// Mitsubishi GX Works2 project: project_cclinkmodules   PLC: Q04UDEH

TYPE D_QJ61BT11N_IN : STRUCT
  x0ModuleError : BOOL;  (* This signal indicates whether the module is normal or faulty,True=Error *)
  x1HostDataOK : BOOL;  (* This signal indicates the data link status of the host station,True=Data Link in Process *)
  x2NotUsed : BOOL;
  x3OtherStLink : BOOL;  (* This signal indicates the data link status of other stations,True= Have Fautly Station *)
  x4NotUsed : BOOL;
  x5NotUsed : BOOL;
  x6NotUsed : BOOL;
  x7NotUsed : BOOL;
  x8NotUsed : BOOL;
  x9NotUsed : BOOL;
  xANotUsed : BOOL;
  xBNotUsed : BOOL;
  xCNotUsed : BOOL;
  xDNotUsed : BOOL;
  xENotUsed : BOOL;
  xFReady : BOOL;  (* This signal indicates whether the module is ready to operate,True=Ready *)
  x10NotUsed : BOOL;
  x11NotUsed : BOOL;
  x12NotUsed : BOOL;
  x13NotUsed : BOOL;
  x14NotUsed : BOOL;
  x15NotUsed : BOOL;
  x16NotUsed : BOOL;
  x17NotUsed : BOOL;
  x18NotUsed : BOOL;
  x19NotUsed : BOOL;
  x1ANotUsed : BOOL;
  x1BNotUsed : BOOL;
  x1CNotUsed : BOOL;
  x1DNotUsed : BOOL;
  x1ENotUsed : BOOL;
  x1FNotUsed : BOOL;
END_STRUCT END_TYPE

TYPE D_Wago_750_325_SystemArea_X : STRUCT
  x0Reserved : BOOL;
  x1Reserved : BOOL;
  x2Reserved : BOOL;
  x3Reserved : BOOL;
  x4Reserved : BOOL;
  x5Reserved : BOOL;
  x6Reserved : BOOL;
  x7Reserved : BOOL;
  x8InitDataReq : BOOL;
  x9InitDataOK : BOOL;
  xAErrorStatus : BOOL;
  xBStationRdy : BOOL;
  xCReserved : BOOL;
  xDReserved : BOOL;
  xEReserved : BOOL;
  xFReserved : BOOL;
END_STRUCT END_TYPE

TYPE D_Wago_750_325_SystemArea_Y : STRUCT
  y0Reserved : BOOL;
  y1Reserved : BOOL;
  y2Reserved : BOOL;
  y3Reserved : BOOL;
  y4Reserved : BOOL;
  y5Reserved : BOOL;
  y6Reserved : BOOL;
  y7Reserved : BOOL;
  y8InitDataComp : BOOL;
  y9InitDataReq : BOOL;
  yAErrorReset : BOOL;
  yBReserved : BOOL;
  yCReserved : BOOL;
  yDReserved : BOOL;
  yEReserved : BOOL;
  yFReserved : BOOL;
END_STRUCT END_TYPE

// global labels: Global1
VAR_GLOBAL
  Module1 : D_QJ61BT11N_IN;
  M_750_325_Sys_x : D_Wago_750_325_SystemArea_X;
  M_750_325_Sys_y : D_Wago_750_325_SystemArea_Y;
  M_750_325_Ch1_x AT X100 : ARRAY [0..7] OF BOOL;
  M_750_325_Ch2_x AT X108 : ARRAY [0..7] OF BOOL;
  M_750_325_Ch1_y AT Y100 : ARRAY [0..7] OF BOOL;
  M_750_325_Ch2_y AT Y108 : ARRAY [0..7] OF BOOL;
END_VAR

// task Task1 (event TRUE, interval 0, priority 31): program1

PROGRAM program1
VAR
  ModuleReady : BOOL;
  WagoCouplerReady : BOOL;
  Wago_750_325_1 : FB_Wago_750_325_HandShake;
  Inited : BOOL;
  Error : BOOL;
  InitError : BOOL;
  Ready : BOOL;
  ModuleError : BOOL;
  Reset : BOOL;
  TON1 : TON;
  iStep : INT;
  Index : INT;
END_VAR

(*Check QJ61BT11N Status *)
	ModuleReady:=Module1.x1HostDataOK AND Module1.xFReady;

(*Check 750-325 Status*)
	WagoCouplerReady:=NOT M_750_325_Sys_x.xAErrorStatus;

Wago_750_325_1(
				io_SystemArea_x:=M_750_325_Sys_x
				,io_SystemArea_y:= M_750_325_Sys_y
				,i_MasterRdy:=ModuleReady
				,i_Reset:=Reset
				,q_Inited:=Inited
				,q_InitError:=InitError
				,q_Ready:=Ready
				,q_ModuleError:=ModuleError
				);
				
CASE iStep OF

	0:
		FOR Index:=0 TO 7 DO
			M_750_325_Ch1_y[Index]:=FALSE;
			M_750_325_Ch2_y[Index]:=TRUE;
		
		END_FOR;
		TON1(
			In:=TRUE
			,PT:=T#1s)
		;
		IF TON1.Q THEN
			TON1(IN:=FALSE);
			iStep:=10;
		END_IF;
		
		
	10:
		FOR Index:=0 TO 7 DO
			M_750_325_Ch1_y[Index]:=TRUE;
			M_750_325_Ch2_y[Index]:=FALSE;
		END_FOR;
				TON1(
			In:=TRUE
			,PT:=T#1s)
		;
		IF TON1.Q THEN
			TON1(IN:=FALSE);
			iStep:=0;
		END_IF;
END_CASE;
END_PROGRAM

FUNCTION_BLOCK FB_Wago_750_325_HandShake
VAR_IN_OUT
  io_SystemArea_x : D_Wago_750_325_SystemArea_X;
  io_SystemArea_y : D_Wago_750_325_SystemArea_Y;
END_VAR
VAR_OUTPUT
  q_ModuleError : BOOL;
  q_Ready : BOOL;
END_VAR
VAR_INPUT
  i_MasterRdy : BOOL;
END_VAR
VAR
  fb_Init_DataReq : R_TRIG;
  iStep : INT;
  TON1 : TON;
END_VAR
VAR_OUTPUT
  q_InitError : BOOL;
END_VAR
VAR_INPUT
  i_Reset : BOOL;
END_VAR
VAR_OUTPUT
  q_Inited : BOOL;
END_VAR



fb_Init_DataReq(
	_CLK:=M_750_325_Sys_x.x8InitDataReq
);

IF fb_Init_DataReq.Q AND i_MasterRdy THEN
	iStep:=1;
END_IF;

CASE iStep OF 
	
	1:
		q_Inited:=FALSE;
		io_SystemArea_y.y8InitDataComp:=TRUE;
		io_SystemArea_y.y9InitDataReq:=TRUE;
		TON1(In:=TRUE,PT:=T#0.5s);
		IF TON1.Q THEN
			iStep:=5;
		END_IF;
	5:
		TON1(in:=FALSE);
		iStep:=10;
	10:
		IF NOT io_SystemArea_x.x8InitDataReq AND io_SystemArea_x.x9InitDataOK THEN
			iStep:=20;
		END_IF;
		IF io_SystemArea_x.xAErrorStatus THEN
			iStep:=99;
		END_IF;
	20:
		io_SystemArea_y.y8InitDataComp:=FALSE;
		io_SystemArea_y.y9InitDataReq:=FALSE;
		iStep:=30;
		TON1(in:=TRUE,pt:=T#0.5s);
		IF TON1.Q THEN
			iStep:=21;
		END_IF;
	21:
		TON1(in:=FALSE);
		iStep:=30;	
	30:
		IF io_SystemArea_x.xBStationRdy THEN
			iStep:=0;
			q_Inited:=TRUE;
		ELSE
			iStep:=99;
		END_IF;
	99:
		q_InitError:=TRUE;
		IF i_Reset THEN
			q_InitError:=FALSE;
			iStep:=0;
		END_IF;				
						
END_CASE;

q_ModuleError:=M_750_325_Sys_x.xAErrorStatus;
q_Ready:=M_750_325_Sys_x.xBStationRdy;
END_FUNCTION_BLOCK
